// TwinCAT 3 PLC project PlcTF6100_OPCUA_Nodeset_Audi
// ProgramVersion: 3.1.4023.0
// libraries:
//   Tc2_Standard, * (Beckhoff Automation GmbH)
//   Tc2_System, * (Beckhoff Automation GmbH)
//   Tc3_Module, * (Beckhoff Automation GmbH)
//   Tc3_OpcUa, * (Beckhoff Automation GmbH)
// project tree:
//   DUTs/ ST_TargetValueType.TcDUT, ST_TimeModelDataType.TcDUT, ST_TargetValueDataType.TcDUT, ST_VersionDataType.TcDUT
//   GVLs/ GVL_Audi_OpcUa.TcGVL
//   Methods/ FB_SetTargetValues.TcPOU, FB_SetTimeModel.TcPOU, FB_Test.TcPOU
//   / PlcTask.TcTTO
//   POUs/ MAIN.TcPOU
// real-time tasks:
//   TASK PlcTask: cycle T#10ms, priority 20, ADS port 350

CONFIGURATION PlcTF6100_OPCUA_Nodeset_Audi
    RESOURCE PLC ON TwinCAT3
        TASK PlcTask(INTERVAL := T#10ms, PRIORITY := 20);
        PROGRAM MAIN WITH PlcTask : MAIN;
    END_RESOURCE
END_CONFIGURATION

// ---- DUTs/ST_TargetValueType.TcDUT
{attribute 'OPC.UA.DA' := '1'}
{attribute 'OPC.UA.DA.StructuredType' := '1'}
{attribute 'pack_mode' := '1'} 
{attribute 'OPC.UA.AdditionalStructuredType.NamespaceName' := 'http://audi.com/OpcUa/CentralIm/'}
{attribute 'OPC.UA.AdditionalStructuredType.Id' := 'i=3010'}
TYPE ST_TargetValueType : UINT; END_TYPE

// ---- DUTs/ST_TimeModelDataType.TcDUT
{attribute 'OPC.UA.DA' := '1'}
{attribute 'OPC.UA.DA.StructuredType' := '1'}
{attribute 'pack_mode' := '1'} 
{attribute 'OPC.UA.AdditionalStructuredType.NamespaceName' := 'http://audi.com/OpcUa/CentralIm/'}
{attribute 'OPC.UA.AdditionalStructuredType.Id' := 'i=3015'}
TYPE ST_TimeModelDataType :
STRUCT
	SwitchingObjectIdentification : BYTE;
	SwitchingObjectNumber : BYTE;
	{attribute 'OPC.UA.DA.Alias' := 'Date'}
	Date1 : DT;
	SwitchingTimes : ARRAY[0..2] OF DINT;
END_STRUCT
END_TYPE

// ---- DUTs/ST_TargetValueDataType.TcDUT
{attribute 'OPC.UA.DA' := '1'}
{attribute 'OPC.UA.DA.StructuredType' := '1'}
{attribute 'pack_mode' := '1'} 
{attribute 'OPC.UA.AdditionalStructuredType.NamespaceName' := 'http://audi.com/OpcUa/CentralIm/'}
{attribute 'OPC.UA.AdditionalStructuredType.Id' := 'i=3011'}
TYPE ST_TargetValueDataType :
STRUCT
	TargetValueType : UINT;
	TargetValue : DINT;
END_STRUCT
END_TYPE

// ---- DUTs/ST_VersionDataType.TcDUT
{attribute 'OPC.UA.DA' := '1'}
{attribute 'OPC.UA.DA.StructuredType' := '1'}
{attribute 'pack_mode' := '1'} 
{attribute 'OPC.UA.AdditionalStructuredType.NamespaceName' := 'http://audi.com/OpcUa/CentralIm/'}
{attribute 'OPC.UA.AdditionalStructuredType.Id' := 'i=3005'}
TYPE ST_VersionDataType :
STRUCT
	Major : UINT;
	Minor : UINT;
	Revision : UINT;
END_STRUCT
END_TYPE

// ---- GVLs/GVL_Audi_OpcUa.TcGVL
{attribute 'qualified_only'}
VAR_GLOBAL
	// ProductionEquipment
	CurrentTimeModel				: ST_TimeModelDataType;
	DeviceManual					: STRING;
	DeviceRevision					: STRING;
	HardwareRevision				: STRING;
	IMVersion						: ST_VersionDataType;
	ItemDesignation					: STRING;
	Manufacturer					: Tc3_OpcUa.UA_LocalizedText;
	Model							: Tc3_OpcUa.UA_LocalizedText;
	NextDayTimeModel				: ST_TimeModelDataType;
	PlcBlockVersion					: ST_VersionDataType;
	RevisionCounter					: DINT;
	SerialNumber					: STRING;
	SerialNumberController			: STRING;
	SerialNumberHW					: STRING;
	SetTargetValues					: FB_SetTargetValues;
	SetTimeModel					: FB_SetTimeModel;
	SoftwareRevision				: STRING;
	TargetValues					: ARRAY[0..2] OF ST_TargetValueDataType;
	//TargetValues					: ARRAY[0..2] OF UINT;
	
	// Diagnostics
	DeviceHealth 					: UINT;
	
	// Eks
	AuthorizationLevel 				: BYTE;
	CostCenter 						: STRING;
	ExpiryDate 						: DT;
	KeyCrc 							: UINT;
	KeyId 							: ULINT;
	OperatorId 						: STRING;
	SafeOperationMode 				: BYTE;
	
	// EnergyData
	ActiveEnergy 					: UDINT;
	ActiveEnergy_EURange			: Tc3_OpcUa.UA_Range;
	ActiveEnergy_StartTimestamp 	: DT;
	ActivePower 					: UDINT;
	ActivePower_EURange				: Tc3_OpcUa.UA_Range;
	
	// ProductionData
	ProductionStatus				: UINT;
	
END_VAR

// ---- POUs/MAIN.TcPOU
PROGRAM MAIN
VAR
	bInit : BOOL := TRUE; // Initializes variables in GVL 	

	{attribute 'OPC.UA.DA' := '1'}
    nCounter1 : INT;
	{attribute 'OPC.UA.DA' := '1'}
    nCounter2 : LREAL;
END_VAR

nCounter1 := nCounter1 + 1;
nCounter2 := nCounter2 + 0.1;

IF bInit THEN
	bInit := FALSE;
	GVL_Audi_OpcUa.CurrentTimeModel.SwitchingObjectIdentification := 1;
	GVL_Audi_OpcUa.CurrentTimeModel.SwitchingObjectNumber := 2;
	GVL_Audi_OpcUa.CurrentTimeModel.Date1 := DT#2020-12-31-23:59:59;
	GVL_Audi_OpcUa.CurrentTimeModel.SwitchingTimes[0] := 0;
	GVL_Audi_OpcUa.CurrentTimeModel.SwitchingTimes[1] := 1;
	GVL_Audi_OpcUa.CurrentTimeModel.SwitchingTimes[2] := 2;
	GVL_Audi_OpcUa.DeviceManual := 'www.beckhoff.com/documentation';
	GVL_Audi_OpcUa.DeviceRevision := 'Revision 42';
	GVL_Audi_OpcUa.HardwareRevision := 'V1.12';
	GVL_Audi_OpcUa.IMVersion.Major := 3;
	GVL_Audi_OpcUa.IMVersion.Minor := 1;
	GVL_Audi_OpcUa.IMVersion.Revision := 4024;
	GVL_Audi_OpcUa.ItemDesignation := 'SomeDesignation';
	GVL_Audi_OpcUa.Manufacturer.sLocaleID := 'en-us';
	GVL_Audi_OpcUa.Manufacturer.sText := 'Beckhoff Automation GmbH & Co. KG';
	GVL_Audi_OpcUa.Model.sLocaleID := 'en-us';
	GVL_Audi_OpcUa.Model.sText := 'CX5140 Embedded Controller';
	GVL_Audi_OpcUa.NextDayTimeModel.SwitchingObjectIdentification := 1;
	GVL_Audi_OpcUa.NextDayTimeModel.SwitchingObjectNumber := 2;
	GVL_Audi_OpcUa.NextDayTimeModel.Date1 := DT#2020-12-31-23:59:59;
	GVL_Audi_OpcUa.NextDayTimeModel.SwitchingTimes[0] := 0;
	GVL_Audi_OpcUa.NextDayTimeModel.SwitchingTimes[1] := 1;
	GVL_Audi_OpcUa.NextDayTimeModel.SwitchingTimes[2] := 2;
	GVL_Audi_OpcUa.PlcBlockVersion.Major := 3;
	GVL_Audi_OpcUa.PlcBlockVersion.Minor := 1;
	GVL_Audi_OpcUa.PlcBlockVersion.Revision := 4024;
	GVL_Audi_OpcUa.RevisionCounter := 42;
	GVL_Audi_OpcUa.SerialNumber := 'V42-42';
	GVL_Audi_OpcUa.SerialNumberController := 'V42-43';
	GVL_Audi_OpcUa.SerialNumberHW := 'V1.1';
	GVL_Audi_OpcUa.SoftwareRevision := 'TwinCAT 3.1 Build 4024.7';
	
	GVL_Audi_OpcUa.DeviceHealth := 2;
	GVL_Audi_OpcUa.AuthorizationLevel := 1;
	GVL_Audi_OpcUa.CostCenter := 'SomeCostCenter';
	GVL_Audi_OpcUa.ExpiryDate := DT#2020-12-31-23:59:59;
	GVL_Audi_OpcUa.KeyCrc := 42;
	GVL_Audi_OpcUa.KeyId := 42;
	GVL_Audi_OpcUa.OperatorId := 'Luke Skywalker';
	GVL_Audi_OpcUa.SafeOperationMode := 2;
	
	GVL_Audi_OpcUa.ActiveEnergy := 42;
	GVL_Audi_OpcUa.ActiveEnergy_EURange.fLow := 0;
	GVL_Audi_OpcUa.ActiveEnergy_EURange.fHigh := 100;
	GVL_Audi_OpcUa.ActiveEnergy_StartTimestamp := DT#2020-01-01-00:00:00;
	
	GVL_Audi_OpcUa.ActivePower := 43;
	GVL_Audi_OpcUa.ActivePower_EURange.fLow := 0;
	GVL_Audi_OpcUa.ActivePower_EURange.fHigh := 100;
	
	GVL_Audi_OpcUa.ProductionStatus := 4; 
	
	GVL_Audi_OpcUa.TargetValues[0].TargetValue := 1;
	GVL_Audi_OpcUa.TargetValues[0].TargetValueType := 1;
	GVL_Audi_OpcUa.TargetValues[1].TargetValue := 1;
	GVL_Audi_OpcUa.TargetValues[1].TargetValueType := 1;
	GVL_Audi_OpcUa.TargetValues[2].TargetValue := 1;
	GVL_Audi_OpcUa.TargetValues[2].TargetValueType := 1;
END_IF

END_PROGRAM

// ---- Methods/FB_SetTargetValues.TcPOU
FUNCTION_BLOCK FB_SetTargetValues
VAR_INPUT
END_VAR
VAR_OUTPUT
END_VAR
VAR
	nCallCount : UINT;
	nTargetValues : ARRAY[0..2] OF ST_TargetValueDataType;
END_VAR

{attribute 'TcRpcEnable' := '1'}
METHOD Abort : HRESULT
VAR_INPUT
END_VAR
END_METHOD

PROPERTY bBusy : BOOL
GET
END_GET
SET
END_SET
END_PROPERTY

{attribute 'TcRpcEnable' := '1'}
METHOD CheckState : HRESULT
VAR_INPUT
	hdl : UDINT;
END_VAR
END_METHOD

PROPERTY hrError : HRESULT
GET
END_GET
SET
END_SET
END_PROPERTY

{attribute 'TcRpcEnable' := '1'}
METHOD Start : HRESULT
VAR_INPUT
	TargetValues : ARRAY[0..2] OF ST_TargetValueDataType;
END_VAR
nCallCount := nCallCount + 1;
nTargetValues[0] := TargetValues[0];
nTargetValues[1] := TargetValues[1];
nTargetValues[2] := TargetValues[2];
END_METHOD

END_FUNCTION_BLOCK

// ---- Methods/FB_SetTimeModel.TcPOU
FUNCTION_BLOCK FB_SetTimeModel
VAR_INPUT
END_VAR
VAR_OUTPUT
END_VAR
VAR
	nCallCount : UINT;
	stTimeModel : ST_TimeModelDataType;
END_VAR

{attribute 'TcRpcEnable' := '1'}
METHOD Abort : HRESULT
VAR_INPUT
END_VAR
END_METHOD

PROPERTY bBusy : BOOL
GET
END_GET
SET
END_SET
END_PROPERTY

{attribute 'TcRpcEnable' := '1'}
METHOD CheckState : HRESULT
VAR_INPUT
	hdl : UDINT;
END_VAR
END_METHOD

PROPERTY hrError : HRESULT
GET
END_GET
SET
END_SET
END_PROPERTY

{attribute 'TcRpcEnable' := '1'}
METHOD Start : HRESULT
VAR_INPUT
	TimeModel : ST_TimeModelDataType;
END_VAR
nCallCount := nCallCount + 1;
stTimeModel := TimeModel;
END_METHOD

END_FUNCTION_BLOCK

// ---- Methods/FB_Test.TcPOU
FUNCTION_BLOCK FB_Test
VAR_INPUT
END_VAR
VAR_OUTPUT
END_VAR
VAR
	nCallCount : UINT;
	nB : ARRAY[0..2] OF INT;
END_VAR

{attribute 'TcRpcEnable' := '1'}
METHOD M_Test : BOOL
VAR_INPUT
	a : INT;
	b : ARRAY[0..2] OF INT;
END_VAR
nCallCount := nCallCount + 1;
nB[0] := b[0];
nB[1] := b[1];
nB[2] := b[2];
M_Test := TRUE;
END_METHOD

END_FUNCTION_BLOCK
